(* PLC project Unnamed, Unknown Unnamed 1 *)
(* stored: creationDateTime 2023-03-18T20:19:53, modificationDateTime 2023-03-18T20:24:31 *)

PROGRAM program0
  VAR_INPUT
    in1 : BOOL;
    in2 : BOOL;
  END_VAR
  VAR_OUTPUT
    out : BOOL;
  END_VAR

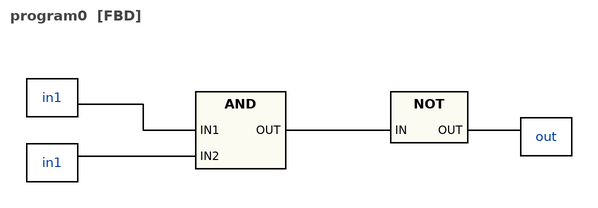
(* FBD diagram, written out as Structured Text *)
out := NOT (in1 AND in1);
END_PROGRAM

CONFIGURATION Config0
  RESOURCE Res0 ON PLC
    TASK task0(INTERVAL := T#20ms, PRIORITY := 0);
    PROGRAM instance0 WITH task0 : program0;
  END_RESOURCE
END_CONFIGURATION
